{attribute 'qualified_only'}
{attribute 'strict'}
{attribute 'to_string'}
TYPE E_DeformationStep :
(
  nothing := 0,
  createdScriptContainer := 1,
  cameraStarted := 2,
  cameraDone := 3,
  gridStarted := 4
);
END_TYPE

(* stored: Version 1.1.0.1, ProductVersion 3.1.4024.11
   EnumerationTextList E_DeformationStep: Id {425d62ec-1999-49f2-9c64-945fc74e4c23} *)
